FUNCTION F_DecreaseTemperature

VAR_INPUT
	stMachine : REFERENCE TO ST_MachineOperatingParameters;
	tCycleTime : REAL;
END_VAR

VAR
END_VAR

stMachine.fTemperature := stMachine.fTemperature - (stMachine.fCoolingConstant * tCycleTime);

END_FUNCTION

(* stored: Version 1.1.0.1, ProductVersion 3.1.4024.12
   POU F_DecreaseTemperature: Id {f05a62f7-741c-47ec-a84f-43983b997651}, SpecialFunc None *)
